// TIA Portal V17 export
// export: Created 2025-03-07T09:16:42.9713385Z, ExportSetting WithDefaults, DisplayName Totally Integrated Automation Portal, DisplayVersion V17 Update 8, DisplayName TIA Portal Openness, DisplayVersion V17 Update 8, DisplayName TIA Portal Version Control Interface, DisplayVersion V17, DisplayName SINAMICS Startdrive Advanced, DisplayVersion V17 SP2, DisplayName SINAMICS Startdrive G110M, G120, G120C, G120D, G120P, G115D, DisplayVersion V17 SP2, DisplayName SINAMICS Startdrive G130, G150, S120, S150, SINAMICS MV, S210, DisplayVersion V17 SP2, DisplayName STEP 7 Professional, DisplayVersion V17 Update 8, DisplayName SINUMERIK ONE STEP 7 Toolbox, DisplayVersion V17 Update 12, DisplayName SINUMERIK 840D sl STEP 7 Toolbox, DisplayVersion V17 Update 12, DisplayName STEP 7 Safety, DisplayVersion V17 Update 6, DisplayName WinCC Advanced, DisplayVersion V17 Update 8
FUNCTION_BLOCK "FB2501_ANALOG_SENSOR"   // FB2501, LAD
{ S7_Optimized_Access := 'FALSE' }
AUTHOR : ETXETAR
VERSION : 1.0
// stored: AutoNumber false, IsIECCheckEnabled false, SetENOAutomatically false, UDAEnableTagReadback false
   VAR_INPUT
      INPUT : Word;   // INPUT
   END_VAR
   VAR_OUTPUT
      CLAMPED_WITHOUT_PART : Bool;   // CLAMPED WITHOUT PARTS / CLAMPED WITHOUT PART
      CLAMPED_WITH_PART : Bool;   // CLAMPED WITH PART
      CLAMPED_STATUS : Bool;   // CLAMPED / CLAMPED STATUS
      UNCLAMPED_STATUS : Bool;   // UNCLAMPED / UNCLAMPED STATUS
   END_VAR
   VAR DB_SPECIFIC
      CURRENT_VALUE { S7_SetPoint := 'True'} : DInt;   // CURRENT VALUE
      CLAMP_MAX_WITHOUT { S7_SetPoint := 'True'} : DInt;   // CLAMP MAX WITHOUT
      CLAMP_MIN_WITHOUT { S7_SetPoint := 'True'} : DInt := DINT#-10000;   // CLAMP MIN WITHOUT
      CLAMP_MAX_WITH { S7_SetPoint := 'True'} : DInt := DINT#-10000;   // CLAMP MAX WITH
      CLAMP_MIN_WITH { S7_SetPoint := 'True'} : DInt := DINT#-10000;   // CLAMP MIN WITH
      UNCLAMP_MAX { S7_SetPoint := 'True'} : DInt := DINT#-10000;   // UNCLAMP MAX
      UNCLAMP_MIN { S7_SetPoint := 'True'} : DInt := DINT#-10000;   // UNCLAMP MIN
      CLAMP_REQUEST { S7_SetPoint := 'True'} : Bool;   // CLAMP REQUEST
      UNCLAMP_REQUEST { S7_SetPoint := 'True'} : Bool;   // UNCLAMP REQUEST
      RELEASE_PRESSURE_REQUEST { S7_SetPoint := 'True'} : Bool;   // PRESSURE RELEASE REQUEST
   END_VAR
BEGIN

REGION Network 1: INPUTS
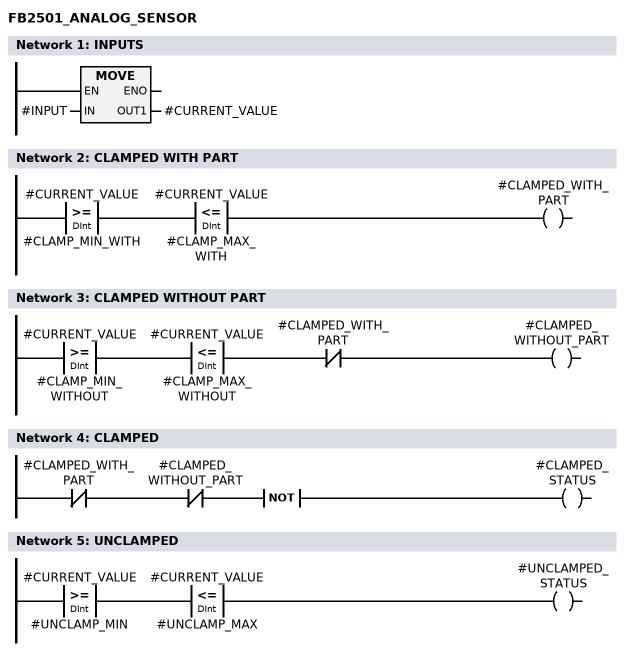
   RUNG wire#powerrail
      { S7_GenerateENO := "TRUE" } Move(in := #INPUT, out1 => #CURRENT_VALUE)
   END_RUNG
   // the same network as SCL:
   #CURRENT_VALUE := #INPUT;
END_REGION

REGION Network 2: CLAMPED WITH PART
   RUNG wire#powerrail
      { S7_Templates := "SrcType := DInt" } GE_Contact(in1 := #CURRENT_VALUE, in2 := #CLAMP_MIN_WITH)
      { S7_Templates := "SrcType := DInt" } LE_Contact(in1 := #CURRENT_VALUE, in2 := #CLAMP_MAX_WITH)
      Coil( #CLAMPED_WITH_PART )
   END_RUNG
   // the same network as SCL:
   #CLAMPED_WITH_PART := (#CURRENT_VALUE >= #CLAMP_MIN_WITH) AND (#CURRENT_VALUE <= #CLAMP_MAX_WITH);
END_REGION

REGION Network 3: CLAMPED WITHOUT PART
   RUNG wire#powerrail
      { S7_Templates := "SrcType := DInt" } GE_Contact(in1 := #CURRENT_VALUE, in2 := #CLAMP_MIN_WITHOUT)
      { S7_Templates := "SrcType := DInt" } LE_Contact(in1 := #CURRENT_VALUE, in2 := #CLAMP_MAX_WITHOUT)
      I_Contact( #CLAMPED_WITH_PART )
      Coil( #CLAMPED_WITHOUT_PART )
   END_RUNG
   // the same network as SCL:
   #CLAMPED_WITHOUT_PART := (#CURRENT_VALUE >= #CLAMP_MIN_WITHOUT) AND (#CURRENT_VALUE <= #CLAMP_MAX_WITHOUT) AND NOT #CLAMPED_WITH_PART;
END_REGION

REGION Network 4: CLAMPED
   RUNG wire#powerrail
      I_Contact( #CLAMPED_WITH_PART )
      I_Contact( #CLAMPED_WITHOUT_PART )
      Not()
      Coil( #CLAMPED_STATUS )
   END_RUNG
   // the same network as SCL:
   #CLAMPED_STATUS := NOT (NOT #CLAMPED_WITH_PART AND NOT #CLAMPED_WITHOUT_PART);
END_REGION

REGION Network 5: UNCLAMPED
   RUNG wire#powerrail
      { S7_Templates := "SrcType := DInt" } GE_Contact(in1 := #CURRENT_VALUE, in2 := #UNCLAMP_MIN)
      { S7_Templates := "SrcType := DInt" } LE_Contact(in1 := #CURRENT_VALUE, in2 := #UNCLAMP_MAX)
      Coil( #UNCLAMPED_STATUS )
   END_RUNG
   // the same network as SCL:
   #UNCLAMPED_STATUS := (#CURRENT_VALUE >= #UNCLAMP_MIN) AND (#CURRENT_VALUE <= #UNCLAMP_MAX);
END_REGION
END_FUNCTION_BLOCK
